FUNCTION_BLOCK PUBLIC FB_LampSetDirectAdapter EXTENDS FB_Lamp
VAR
	fbLampSetDirect		: FB_LampSetDirect;
END_VAR

// Reduces the control value by 5 in the range of 10 to 100.
METHOD PUBLIC DimDown
IF (fbLampSetDirect.nLightLevel >= 15) THEN
	fbLampSetDirect.SetLightLevel(fbLampSetDirect.nLightLevel - 5);
END_IF
IF (_ipObserver <> 0) THEN
	_ipObserver.Update(fbLampSetDirect.nLightLevel);
END_IF
END_METHOD

// Increments the control value by 5 in the range of 10 to 100.
METHOD PUBLIC DimUp
IF (fbLampSetDirect.nLightLevel <= 95) THEN
	fbLampSetDirect.SetLightLevel(fbLampSetDirect.nLightLevel + 5);
END_IF
IF (_ipObserver <> 0) THEN
	_ipObserver.Update(fbLampSetDirect.nLightLevel);
END_IF
END_METHOD

// Sets the control value to 0.
METHOD PUBLIC Off
fbLampSetDirect.SetLightLevel(0);
IF (_ipObserver <> 0) THEN
	_ipObserver.Update(fbLampSetDirect.nLightLevel);
END_IF
END_METHOD

// Sets the control value to 100.
METHOD PUBLIC On
fbLampSetDirect.SetLightLevel(100);
IF (_ipObserver <> 0) THEN
	_ipObserver.Update(fbLampSetDirect.nLightLevel);
END_IF
END_METHOD

END_FUNCTION_BLOCK

(* stored: Version 1.1.0.1, ProductVersion 3.1.4024.11
   POU FB_LampSetDirectAdapter: Id {b43edb15-db5d-436e-adda-e04f3d808833}, SpecialFunc None
   Method DimDown: Id {104dfa9e-d922-4c45-bf9f-4ec89df56551}
   Method DimUp: Id {eaa7b6f8-3f10-4d48-b412-2bbd0af95e7b}
   Method Off: Id {03cb4157-9aba-43a4-8729-d4e37e60b528}
   Method On: Id {743aa10c-6d50-4098-84b2-dc39575e8414} *)
